// LS Electric XG5000 project: 333
// PLC LSPLC
// module base 0 slot 0: 입출력 모듈:XBM-DN32H (DC 24V입력/TR 출력, 32점)

PROGRAM NewProgram (task: 스캔 프로그램)

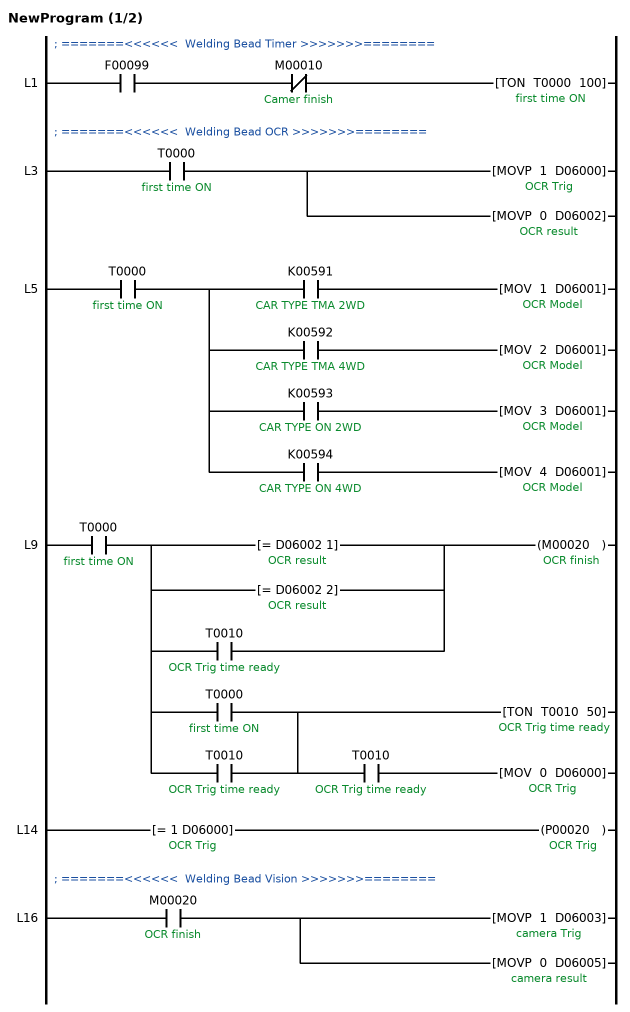
// =======<<<<<<  Welding Bead Timer >>>>>>>========
; L1
LOAD      F00099
AND NOT   M00010	// Camer finish
TON       T0000 100	// first time ON
// =======<<<<<<  Welding Bead OCR >>>>>>>========
; L3
LOAD      T0000	// first time ON
MOVP      1 D06000	// OCR Trig
MOVP      0 D06002	// OCR result
; L5
LOAD      T0000	// first time ON
MPUSH
AND       K00591	// CAR TYPE TMA 2WD
MOV       1 D06001	// OCR Model
MLOAD
AND       K00592	// CAR TYPE TMA 4WD
MOV       2 D06001	// OCR Model
MLOAD
AND       K00593	// CAR TYPE ON 2WD
MOV       3 D06001	// OCR Model
MPOP
AND       K00594	// CAR TYPE ON 4WD
MOV       4 D06001	// OCR Model
; L9
LOAD      T0000	// first time ON
MPUSH
LOAD=     D06002 1	// OCR result
OR=       D06002 2	// OCR result
OR        T0010	// OCR Trig time ready
AND LOAD
OUT       M00020	// OCR finish
MPOP
LOAD      T0000	// first time ON
OR        T0010	// OCR Trig time ready
AND LOAD
TON       T0010 50	// OCR Trig time ready
AND       T0010	// OCR Trig time ready
MOV       0 D06000	// OCR Trig
; L14
LOAD=     1 D06000	// OCR Trig
OUT       P00020	// OCR Trig
// =======<<<<<<  Welding Bead Vision >>>>>>>========
; L16
LOAD      M00020	// OCR finish
MOVP      1 D06003	// camera Trig
MOVP      0 D06005	// camera result

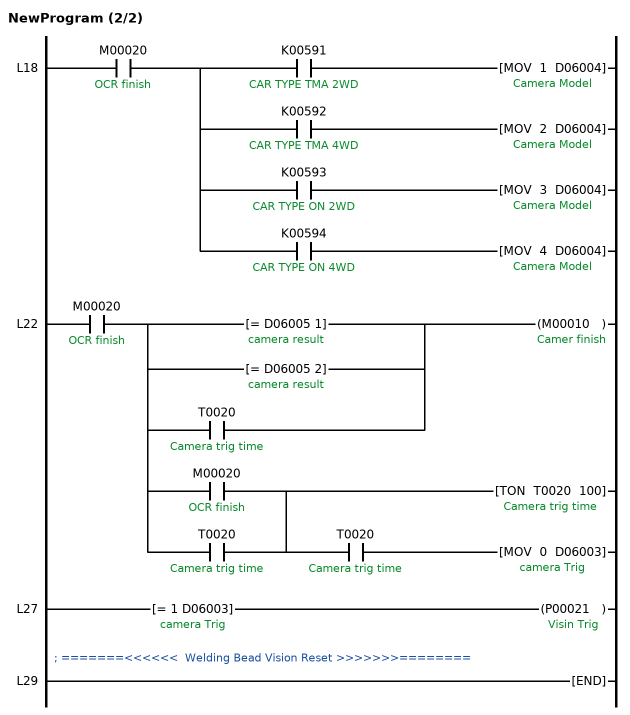
; L18
LOAD      M00020	// OCR finish
MPUSH
AND       K00591	// CAR TYPE TMA 2WD
MOV       1 D06004	// Camera Model
MLOAD
AND       K00592	// CAR TYPE TMA 4WD
MOV       2 D06004	// Camera Model
MLOAD
AND       K00593	// CAR TYPE ON 2WD
MOV       3 D06004	// Camera Model
MPOP
AND       K00594	// CAR TYPE ON 4WD
MOV       4 D06004	// Camera Model
; L22
LOAD      M00020	// OCR finish
MPUSH
LOAD=     D06005 1	// camera result
OR=       D06005 2	// camera result
OR        T0020	// Camera trig time
AND LOAD
OUT       M00010	// Camer finish
MPOP
LOAD      M00020	// OCR finish
OR        T0020	// Camera trig time
AND LOAD
TON       T0020 100	// Camera trig time
AND       T0020	// Camera trig time
MOV       0 D06003	// camera Trig
; L27
LOAD=     1 D06003	// camera Trig
OUT       P00021	// Visin Trig
// =======<<<<<<  Welding Bead Vision Reset >>>>>>>========
; L29
END

VARIABLES AND COMMENTS (devices not used above)
D06006	WORD	Vision Ready
T0001	BIT/WORD	Welding Bead Trig ON
T0002	BIT/WORD	Trig OFF
T0030	BIT/WORD	Camera finish time 
T0005	BIT/WORD	Reset time